Fanuc TP program (LS listing): JOB_VAR_COMMON.LS

/PROG  JOB_VAR_COMMON
/ATTR
OWNER		= MNEDITOR;
COMMENT		= "";
PROG_SIZE	= 43409;
CREATE		= DATE 19-03-19  TIME 16:19:56;
MODIFIED	= DATE 26-05-22  TIME 14:18:32;
FILE_NAME	= JOB_VAR_;
VERSION		= 0;
LINE_COUNT	= 1720;
MEMORY_SIZE	= 43957;
PROTECT		= READ_WRITE;
TCD:  STACK_SIZE	= 0,
      TASK_PRIORITY	= 50,
      TIME_SLICE	= 0,
      BUSY_LAMP_OFF	= 0,
      ABORT_REQUEST	= 0,
      PAUSE_REQUEST	= 0;
DEFAULT_GROUP	= 1,*,*,*,*;
CONTROL_CODE	= 00000000 00000000;
/APPL

AUTO_SINGULARITY_HEADER;
  ENABLE_SINGULARITY_AVOIDANCE   : TRUE;
/MN
   1:  !This is the common point ;
   2:  !template, all points are ;
   3:  !same if concentric ;
   4:  !---------------------------- ;
   5:  !Assign variable point profile ;
   6:  R[103]=AR[1]    ;
   7:  !--------------------------- ;
   8:  !SR[1] = "JOB_VAR_ID_GRIP" ;
   9:  !R[103]=100 -> "JOB_VAR_ID_GRIP" ;
  10:  !---------------------------- ;
  11:  !2By3 INF ID-GRIP, Max 18 piece ;
  12:  !Straight Face-plate Up/Down Pick ;
  13:  !---------------------------- ;
  14:  SELECT R[103]=100,JMP LBL[100] ;
  15:  !---------------------------- ;
  16:  !2By3 INF ID-GRIP, 45Deg Shift ;
  17:  !J4 Shift to Diagonal Pick ;
  18:         =110,JMP LBL[110] ;
  19:  !---------------------------- ;
  20:  !3By4 INF Sheet, Max 36 piece ;
  21:  !Straight Face-plate Up/Down Pick ;
  22:         =150,JMP LBL[150] ;
  23:  !---------------------------- ;
  24:  !3By4 INF Sheet, metal plate Max ;
  25:  !Straight Face-plate Up/Down Pick ;
  26:         =160,JMP LBL[160] ;
  27:  !---------------------------- ;
  28:  !3By4 INF Sheet, Max 72 piece ;
  29:  !Straight Face-plate Up/Down Pick ;
  30:         =170,JMP LBL[170] ;
  31:  !---------------------------- ;
  32:  !SR[2] = "JOB_VAR_OD_GRIP" ;
  33:  !R[103]=200 -> "JOB_VAR_OD_GRIP" ;
  34:  !---------------------------- ;
  35:  !2By3 INF OD-GRIP, Max 18 piece ;
  36:  !Straight Face-plate Up/Down Pick ;
  37:         =200,JMP LBL[200] ;
  38:  !---------------------------- ;
  39:  !2By3 INF OD-GRIP, 45Deg Shift ;
  40:  !J4 Shift to Diagonal Pick ;
  41:         =210,JMP LBL[210] ;
  42:  !---------------------------- ;
  43:  !3By4 INF OD-GRIP, Max 36 piece ;
  44:  !Straight Face-plate Up/Down Pick ;
  45:         =250,JMP LBL[250] ;
  46:  !---------------------------- ;
  47:  !3By4 INF OD-GRIP, 45Deg Shift ;
  48:  !J4 Shift to Diagonal Pick ;
  49:         =260,JMP LBL[260] ;
  50:  !---------------------------- ;
  51:  !4By6 INF OD-GRIP, Max 144 piece ;
  52:  !6By9 OFT 3 Tray ;
  53:         =270,JMP LBL[270] ;
  54:  !---------------------------- ;
  55:  !4By6 INF OD-GRIP, Max 144 piece ;
  56:  !6By8 OFT 3 Tray ;
  57:         =280,JMP LBL[280] ;
  58:  !---------------------------- ;
  59:  !Bar Feed OFT only, Max 144 piece ;
  60:  !4By9 OFT 4 Tray ;
  61:         =300,JMP LBL[300] ;
  62:  !---------------------------- ;
  63:  !Bar Feed OFT only, Max 144 piece ;
  64:  !6By8 OFT 3 Tray ;
  65:         =320,JMP LBL[320] ;
  66:  !---------------------------- ;
  67:  !3By4 INF Box ;
  68:  !Straight Up/Down Pick ;
  69:         =340,JMP LBL[340] ;
  70:  !---------------------------- ;
  71:  LBL[100] ;
  72:  !---------------------------- ;
  73:  !R[103]=100 -> "JOB_VAR_ID_GRIP" ;
  74:  !2By3 INF ID-GRIP, Max 18 piece ;
  75:  !Straight Face-plate Up/Down Pick ;
  76:  !---------------------------- ;
  77:  !Built PR[40] as Infeed P[1] ;
  78:  R[200]=40    ;
  79:   ;
  80:  R[201]=120.088    ;
  81:  R[202]=782.289    ;
  82:  R[203]=500.058    ;
  83:  R[204]=(-150.905)    ;
  84:  R[205]=(-89.467)    ;
  85:  R[206]=(-28.099)    ;
  86:   ;
  87:  CALL CREATE_PR(R[200],R[201],R[202],R[203],R[204],R[205],R[206]) ;
  88:   ;
  89:  !---------------------------- ;
  90:  !R[103]=100 -> "JOB_VAR_ID_GRIP" ;
  91:  !2By3 INF ID-GRIP, Max 18 piece ;
  92:  !Straight Face-plate Up/Down Pick ;
  93:  !---------------------------- ;
  94:  !Built PR[41] as Infeed P[2] ;
  95:  R[210]=41    ;
  96:   ;
  97:  R[211]=120.251    ;
  98:  R[212]=334.967    ;
  99:  R[213]=500.04    ;
 100:  R[214]=(-147.763)    ;
 101:  R[215]=(-89.089)    ;
 102:  R[216]=(-31.313)    ;
 103:   ;
 104:  CALL CREATE_PR(R[210],R[211],R[212],R[213],R[214],R[215],R[216]) ;
 105:   ;
 106:  !---------------------------- ;
 107:  !R[103]=100 -> "JOB_VAR_ID_GRIP" ;
 108:  !2By3 INF ID-GRIP, Max 18 piece ;
 109:  !Straight Face-plate Up/Down Pick ;
 110:  !---------------------------- ;
 111:  !Built PR[42] as Infeed P[3] ;
 112:  R[220]=42    ;
 113:   ;
 114:  R[221]=118.765    ;
 115:  R[222]=(-120.642)    ;
 116:  R[223]=500.756    ;
 117:  R[224]=(-153.606)    ;
 118:  R[225]=(-89.098)    ;
 119:  R[226]=(-25.398)    ;
 120:   ;
 121:  CALL CREATE_PR(R[220],R[221],R[222],R[223],R[224],R[225],R[226]) ;
 122:   ;
 123:  !---------------------------- ;
 124:  !R[103]=100 -> "JOB_VAR_ID_GRIP" ;
 125:  !2By3 INF ID-GRIP, Max 18 piece ;
 126:  !Straight Face-plate Up/Down Pick ;
 127:  !---------------------------- ;
 128:  !Built PR[50] as Outfeed P[1] ;
 129:  R[230]=50    ;
 130:   ;
 131:  R[231]=110.122    ;
 132:  R[232]=(-117.756)    ;
 133:  R[233]=500    ;
 134:  R[234]=6.053    ;
 135:  R[235]=(-88.646)    ;
 136:  R[236]=173.167    ;
 137:   ;
 138:  CALL CREATE_PR(R[230],R[231],R[232],R[233],R[234],R[235],R[236]) ;
 139:   ;
 140:  !---------------------------- ;
 141:  !R[103]=100 -> "JOB_VAR_ID_GRIP" ;
 142:  !2By3 INF ID-GRIP, Max 18 piece ;
 143:  !Straight Face-plate Up/Down Pick ;
 144:  !---------------------------- ;
 145:  !Built PR[51] as Outfeed P[2] ;
 146:  R[240]=51    ;
 147:   ;
 148:  R[241]=113.046    ;
 149:  R[242]=333.772    ;
 150:  R[243]=500    ;
 151:  R[244]=5.59    ;
 152:  R[245]=(-88.801)    ;
 153:  R[246]=173.593    ;
 154:   ;
 155:  CALL CREATE_PR(R[240],R[241],R[242],R[243],R[244],R[245],R[246]) ;
 156:   ;
 157:  !---------------------------- ;
 158:  !R[103]=100 -> "JOB_VAR_ID_GRIP" ;
 159:  !2By3 INF ID-GRIP, Max 18 piece ;
 160:  !Straight Face-plate Up/Down Pick ;
 161:  !---------------------------- ;
 162:  !Built PR[52] as Outfeed P[3] ;
 163:  R[250]=52    ;
 164:   ;
 165:  R[251]=115.343    ;
 166:  R[252]=785.028    ;
 167:  R[253]=500    ;
 168:  R[254]=(-7.342)    ;
 169:  R[255]=(-88.924)    ;
 170:  R[256]=(-173.386)    ;
 171:   ;
 172:  CALL CREATE_PR(R[250],R[251],R[252],R[253],R[254],R[255],R[256]) ;
 173:   ;
 174:  !Jump to end of the program ;
 175:  JMP LBL[9999] ;
 176:  !Template Ends ;
 177:   ;
 178:  !---------------------------- ;
 179:  LBL[110] ;
 180:  !---------------------------- ;
 181:  !R[103]=110 -> "JOB_VAR_ID_GRIP" ;
 182:  !2By3 INF ID-GRIP, 45Deg Shift ;
 183:  !J4 Shift to Diagonal Pick ;
 184:  !---------------------------- ;
 185:  !2By3 INF ID-GRIP, Max 18 piece ;
 186:  !---------------------------- ;
 187:  !Built PR[40] as Infeed P[1] ;
 188:  R[200]=40    ;
 189:   ;
 190:  R[201]=112.509    ;
 191:  R[202]=779.307    ;
 192:  R[203]=300    ;
 193:  R[204]=148.582    ;
 194:  R[205]=(-89.868)    ;
 195:  R[206]=(-7.553)    ;
 196:   ;
 197:  CALL CREATE_PR(R[200],R[201],R[202],R[203],R[204],R[205],R[206]) ;
 198:   ;
 199:  !---------------------------- ;
 200:  !R[103]=110 -> "JOB_VAR_ID_GRIP" ;
 201:  !2By3 INF ID-GRIP, 45Deg Shift ;
 202:  !J4 Shift to Diagonal Pick ;
 203:  !---------------------------- ;
 204:  !Built PR[41] as Infeed P[2] ;
 205:  R[210]=41    ;
 206:   ;
 207:  R[211]=112.917    ;
 208:  R[212]=329.437    ;
 209:  R[213]=300    ;
 210:  R[214]=157.871    ;
 211:  R[215]=(-89.833)    ;
 212:  R[216]=(-16.841)    ;
 213:   ;
 214:  CALL CREATE_PR(R[210],R[211],R[212],R[213],R[214],R[215],R[216]) ;
 215:   ;
 216:  !---------------------------- ;
 217:  !R[103]=110 -> "JOB_VAR_ID_GRIP" ;
 218:  !2By3 INF ID-GRIP, 45Deg Shift ;
 219:  !J4 Shift to Diagonal Pick ;
 220:  !---------------------------- ;
 221:  !Built PR[42] as Infeed P[3] ;
 222:  R[220]=42    ;
 223:   ;
 224:  R[221]=112.976    ;
 225:  R[222]=(-121.647)    ;
 226:  R[223]=300    ;
 227:  R[224]=162.478    ;
 228:  R[225]=(-89.805)    ;
 229:  R[226]=(-21.447)    ;
 230:   ;
 231:  CALL CREATE_PR(R[220],R[221],R[222],R[223],R[224],R[225],R[226]) ;
 232:   ;
 233:  !---------------------------- ;
 234:  !R[103]=110 -> "JOB_VAR_ID_GRIP" ;
 235:  !2By3 INF ID-GRIP, 45Deg Shift ;
 236:  !J4 Shift to Diagonal Drop ;
 237:  !---------------------------- ;
 238:  !Built PR[50] as OTF P[1] ;
 239:  R[230]=50    ;
 240:   ;
 241:  R[231]=110.895    ;
 242:  R[232]=(-123.626)    ;
 243:  R[233]=300    ;
 244:  R[234]=155.317    ;
 245:  R[235]=(-89.484)    ;
 246:  R[236]=(-24.715)    ;
 247:   ;
 248:  CALL CREATE_PR(R[230],R[231],R[232],R[233],R[234],R[235],R[236]) ;
 249:   ;
 250:  !---------------------------- ;
 251:  !R[103]=110 -> "JOB_VAR_ID_GRIP" ;
 252:  !2By3 INF ID-GRIP, 45Deg Shift ;
 253:  !J4 Shift to Diagonal Drop ;
 254:  !---------------------------- ;
 255:  !Built PR[51] as OTF P[2] ;
 256:  R[240]=51    ;
 257:   ;
 258:  R[241]=112.415    ;
 259:  R[242]=326.508    ;
 260:  R[243]=300    ;
 261:  R[244]=156.037    ;
 262:  R[245]=(-89.475)    ;
 263:  R[246]=(-25.441)    ;
 264:   ;
 265:  CALL CREATE_PR(R[240],R[241],R[242],R[243],R[244],R[245],R[246]) ;
 266:   ;
 267:  !---------------------------- ;
 268:  !R[103]=110 -> "JOB_VAR_ID_GRIP" ;
 269:  !2By3 INF ID-GRIP, 45Deg Shift ;
 270:  !J4 Shift to Diagonal Drop ;
 271:  !---------------------------- ;
 272:  !Built PR[52] as OTF P[3] ;
 273:  R[250]=52    ;
 274:   ;
 275:  R[251]=113.171    ;
 276:  R[252]=777.28    ;
 277:  R[253]=300    ;
 278:  R[254]=155.207    ;
 279:  R[255]=(-89.455)    ;
 280:  R[256]=(-24.623)    ;
 281:   ;
 282:  CALL CREATE_PR(R[250],R[251],R[252],R[253],R[254],R[255],R[256]) ;
 283:   ;
 284:  !Jump to end of the program ;
 285:  JMP LBL[9999] ;
 286:  !Template Ends ;
 287:   ;
 288:  !---------------------------- ;
 289:  LBL[150] ;
 290:  !---------------------------- ;
 291:  !R[103]=150 -> "JOB_VAR_ID_GRIP" ;
 292:  !3By4 INF Sheet, Max 36 piece ;
 293:  !Straight Face-plate Up/Down Pick ;
 294:  !---------------------------- ;
 295:  !Built PR[40] as Infeed P[1] ;
 296:  R[200]=40    ;
 297:   ;
 298:  R[201]=69.764    ;
 299:  R[202]=828.432    ;
 300:  R[203]=300    ;
 301:  R[204]=(-158.565)    ;
 302:  R[205]=(-89.413)    ;
 303:  R[206]=(-20.581)    ;
 304:   ;
 305:  CALL CREATE_PR(R[200],R[201],R[202],R[203],R[204],R[205],R[206]) ;
 306:   ;
 307:  !---------------------------- ;
 308:  !R[103]=150 -> "JOB_VAR_ID_GRIP" ;
 309:  !Straight Up/Down Pick ;
 310:  !3By4 INF Sheet, Max 36 piece ;
 311:  !---------------------------- ;
 312:  !Built PR[41] as Infeed P[2] ;
 313:  R[210]=41    ;
 314:   ;
 315:  R[211]=72.484    ;
 316:  R[212]=376.905    ;
 317:  R[213]=300    ;
 318:  R[214]=(-149.34)    ;
 319:  R[215]=(-89.283)    ;
 320:  R[216]=(-29.779)    ;
 321:   ;
 322:  CALL CREATE_PR(R[210],R[211],R[212],R[213],R[214],R[215],R[216]) ;
 323:   ;
 324:  !---------------------------- ;
 325:  !R[103]=150 -> "JOB_VAR_ID_GRIP" ;
 326:  !3By4 INF Sheet, Max 36 piece ;
 327:  !Straight Face-plate Up/Down Pick ;
 328:  !---------------------------- ;
 329:  !Built PR[42] as Infeed P[3] ;
 330:  R[220]=42    ;
 331:   ;
 332:  R[221]=73.047    ;
 333:  R[222]=(-73.901)    ;
 334:  R[223]=300    ;
 335:  R[224]=(-162.774)    ;
 336:  R[225]=(-88.893)    ;
 337:  R[226]=(-16.221)    ;
 338:   ;
 339:  CALL CREATE_PR(R[220],R[221],R[222],R[223],R[224],R[225],R[226]) ;
 340:   ;
 341:  !---------------------------- ;
 342:  !R[103]=150 -> "JOB_VAR_ID_GRIP" ;
 343:  !3By4 INF Sheet, Max 36 piece ;
 344:  !Straight Face-plate Up/Down Pick ;
 345:  !---------------------------- ;
 346:  !Built PR[50] as OTF P[1] ;
 347:  R[230]=50    ;
 348:   ;
 349:  R[231]=66.596    ;
 350:  R[232]=(-72.932)    ;
 351:  R[233]=300    ;
 352:  R[234]=5.353    ;
 353:  R[235]=(-88.806)    ;
 354:  R[236]=173.83    ;
 355:   ;
 356:  CALL CREATE_PR(R[230],R[231],R[232],R[233],R[234],R[235],R[236]) ;
 357:   ;
 358:  !---------------------------- ;
 359:  !R[103]=150 -> "JOB_VAR_ID_GRIP" ;
 360:  !3By4 INF Sheet, Max 36 piece ;
 361:  !Straight Face-plate Up/Down Pick ;
 362:  !---------------------------- ;
 363:  !Built PR[51] as OTF P[2] ;
 364:  R[240]=51    ;
 365:   ;
 366:  R[241]=70.095    ;
 367:  R[242]=378.905    ;
 368:  R[243]=300    ;
 369:  R[244]=(-4.178)    ;
 370:  R[245]=(-88.742)    ;
 371:  R[246]=(-176.605)    ;
 372:   ;
 373:  CALL CREATE_PR(R[240],R[241],R[242],R[243],R[244],R[245],R[246]) ;
 374:   ;
 375:  !---------------------------- ;
 376:  !R[103]=150 -> "JOB_VAR_ID_GRIP" ;
 377:  !3By4 INF Sheet, Max 36 piece ;
 378:  !Straight Face-plate Up/Down Pick ;
 379:  !---------------------------- ;
 380:  !Built PR[52] as OTF P[3] ;
 381:  R[250]=52    ;
 382:   ;
 383:  R[251]=70.211    ;
 384:  R[252]=829.862    ;
 385:  R[253]=300    ;
 386:  R[254]=(-7.014)    ;
 387:  R[255]=(-88.859)    ;
 388:  R[256]=(-173.67)    ;
 389:   ;
 390:  CALL CREATE_PR(R[250],R[251],R[252],R[253],R[254],R[255],R[256]) ;
 391:   ;
 392:  !Jump to end of the program ;
 393:  JMP LBL[9999] ;
 394:  !Template Ends ;
 395:   ;
 396:  !---------------------------- ;
 397:  LBL[160] ;
 398:  !---------------------------- ;
 399:  !R[103]=160 -> "JOB_VAR_ID_GRIP" ;
 400:  !3By4 INF Sheet, metal plate Max ;
 401:  !Straight Face-plate Up/Down Pick ;
 402:  !---------------------------- ;
 403:  !Built PR[40] as Infeed P[1] ;
 404:  R[200]=40    ;
 405:   ;
 406:  R[201]=78.195    ;
 407:  R[202]=824.843    ;
 408:  R[203]=300    ;
 409:  R[204]=(-.36)    ;
 410:  R[205]=(-88.464)    ;
 411:  R[206]=(-178.776)    ;
 412:   ;
 413:  CALL CREATE_PR(R[200],R[201],R[202],R[203],R[204],R[205],R[206]) ;
 414:   ;
 415:  !---------------------------- ;
 416:  !R[103]=160 -> "JOB_VAR_ID_GRIP" ;
 417:  !3By4 INF Sheet, metal plate Max ;
 418:  !Straight Face-plate Up/Down Pick ;
 419:  !---------------------------- ;
 420:  !Built PR[41] as Infeed P[2] ;
 421:  R[210]=41    ;
 422:   ;
 423:  R[211]=75.096    ;
 424:  R[212]=376.135    ;
 425:  R[213]=300    ;
 426:  R[214]=24.515    ;
 427:  R[215]=(-88.736)    ;
 428:  R[216]=156.675    ;
 429:   ;
 430:  CALL CREATE_PR(R[210],R[211],R[212],R[213],R[214],R[215],R[216]) ;
 431:   ;
 432:  !---------------------------- ;
 433:  !R[103]=160 -> "JOB_VAR_ID_GRIP" ;
 434:  !3By4 INF Sheet, metal plate Max ;
 435:  !Straight Face-plate Up/Down Pick ;
 436:  !---------------------------- ;
 437:  !Built PR[42] as Infeed P[3] ;
 438:  R[220]=42    ;
 439:   ;
 440:  R[221]=72.884    ;
 441:  R[222]=(-76.019)    ;
 442:  R[223]=300    ;
 443:  R[224]=(-1.211)    ;
 444:  R[225]=(-88.387)    ;
 445:  R[226]=(-177.625)    ;
 446:   ;
 447:  CALL CREATE_PR(R[220],R[221],R[222],R[223],R[224],R[225],R[226]) ;
 448:   ;
 449:  !---------------------------- ;
 450:  !R[103]=160 -> "JOB_VAR_ID_GRIP" ;
 451:  !3By4 INF Sheet, metal plate Max ;
 452:  !Straight Face-plate Up/Down Pick ;
 453:  !---------------------------- ;
 454:  !Built PR[50] as OTF P[1] ;
 455:  R[230]=50    ;
 456:   ;
 457:  R[231]=66.596    ;
 458:  R[232]=(-72.932)    ;
 459:  R[233]=700    ;
 460:  R[234]=5.353    ;
 461:  R[235]=(-88.806)    ;
 462:  R[236]=173.83    ;
 463:   ;
 464:  CALL CREATE_PR(R[230],R[231],R[232],R[233],R[234],R[235],R[236]) ;
 465:   ;
 466:  !---------------------------- ;
 467:  !R[103]=160 -> "JOB_VAR_ID_GRIP" ;
 468:  !3By4 INF Sheet, metal plate Max ;
 469:  !Straight Face-plate Up/Down Pick ;
 470:  !---------------------------- ;
 471:  !Built PR[51] as OTF P[2] ;
 472:  R[240]=51    ;
 473:   ;
 474:  R[241]=70.095    ;
 475:  R[242]=378.905    ;
 476:  R[243]=700    ;
 477:  R[244]=(-4.178)    ;
 478:  R[245]=(-88.742)    ;
 479:  R[246]=(-176.605)    ;
 480:   ;
 481:  CALL CREATE_PR(R[240],R[241],R[242],R[243],R[244],R[245],R[246]) ;
 482:   ;
 483:  !---------------------------- ;
 484:  !R[103]=160 -> "JOB_VAR_ID_GRIP" ;
 485:  !3By4 INF Sheet, metal plate Max ;
 486:  !Straight Face-plate Up/Down Pick ;
 487:  !---------------------------- ;
 488:  !Built PR[52] as OTF P[3] ;
 489:  R[250]=52    ;
 490:   ;
 491:  R[251]=70.211    ;
 492:  R[252]=829.862    ;
 493:  R[253]=700    ;
 494:  R[254]=(-7.014)    ;
 495:  R[255]=(-88.859)    ;
 496:  R[256]=(-173.67)    ;
 497:   ;
 498:  CALL CREATE_PR(R[250],R[251],R[252],R[253],R[254],R[255],R[256]) ;
 499:   ;
 500:  !Jump to end of the program ;
 501:  JMP LBL[9999] ;
 502:  !Template Ends ;
 503:   ;
 504:  !---------------------------- ;
 505:  LBL[170] ;
 506:  !---------------------------- ;
 507:  !R[103]=170 -> "JOB_VAR_ID_GRIP" ;
 508:  !3By4 INF Sheet, Max 72 piece ;
 509:  !Straight Face-plate Up/Down Pick ;
 510:  !---------------------------- ;
 511:  !Built PR[40] as Infeed P[1] ;
 512:  R[200]=40    ;
 513:   ;
 514:  R[201]=70.947    ;
 515:  R[202]=827.937    ;
 516:  R[203]=300    ;
 517:  R[204]=19.09    ;
 518:  R[205]=(-88.606)    ;
 519:  R[206]=161.741    ;
 520:   ;
 521:  CALL CREATE_PR(R[200],R[201],R[202],R[203],R[204],R[205],R[206]) ;
 522:   ;
 523:  !---------------------------- ;
 524:  !R[103]=170 -> "JOB_VAR_ID_GRIP" ;
 525:  !3By4 INF Sheet, Max 72 piece ;
 526:  !Straight Face-plate Up/Down Pick ;
 527:  !---------------------------- ;
 528:  !Built PR[41] as Infeed P[2] ;
 529:  R[210]=41    ;
 530:   ;
 531:  R[211]=69.577    ;
 532:  R[212]=378.246    ;
 533:  R[213]=300    ;
 534:  R[214]=19.393    ;
 535:  R[215]=(-88.529)    ;
 536:  R[216]=161.453    ;
 537:   ;
 538:  CALL CREATE_PR(R[210],R[211],R[212],R[213],R[214],R[215],R[216]) ;
 539:   ;
 540:  !---------------------------- ;
 541:  !R[103]=170 -> "JOB_VAR_ID_GRIP" ;
 542:  !3By4 INF Sheet, Max 72 piece ;
 543:  !Straight Face-plate Up/Down Pick ;
 544:  !---------------------------- ;
 545:  !Built PR[42] as Infeed P[3] ;
 546:  R[220]=42    ;
 547:   ;
 548:  R[221]=67.051    ;
 549:  R[222]=(-70.861)    ;
 550:  R[223]=300    ;
 551:  R[224]=17.005    ;
 552:  R[225]=(-88.405)    ;
 553:  R[226]=163.867    ;
 554:   ;
 555:  CALL CREATE_PR(R[220],R[221],R[222],R[223],R[224],R[225],R[226]) ;
 556:   ;
 557:  !---------------------------- ;
 558:  !R[103]=170 -> "JOB_VAR_ID_GRIP" ;
 559:  !3By4 INF Sheet, Max 72 piece ;
 560:  !Straight Face-plate Up/Down Pick ;
 561:  !---------------------------- ;
 562:  !Built PR[46] as Infeed P[4] ;
 563:  R[230]=46    ;
 564:   ;
 565:  R[231]=66.596    ;
 566:  R[232]=(-72.932)    ;
 567:  R[233]=300    ;
 568:  R[234]=5.353    ;
 569:  R[235]=(-88.806)    ;
 570:  R[236]=173.83    ;
 571:   ;
 572:  CALL CREATE_PR(R[230],R[231],R[232],R[233],R[234],R[235],R[236]) ;
 573:   ;
 574:  !---------------------------- ;
 575:  !R[103]=170 -> "JOB_VAR_ID_GRIP" ;
 576:  !3By4 INF Sheet, Max 72 piece ;
 577:  !Straight Face-plate Up/Down Pick ;
 578:  !---------------------------- ;
 579:  !Built PR[47] as Infeed P[5] ;
 580:  R[240]=47    ;
 581:   ;
 582:  R[241]=70.095    ;
 583:  R[242]=378.905    ;
 584:  R[243]=300    ;
 585:  R[244]=(-4.178)    ;
 586:  R[245]=(-88.742)    ;
 587:  R[246]=(-176.605)    ;
 588:   ;
 589:  CALL CREATE_PR(R[240],R[241],R[242],R[243],R[244],R[245],R[246]) ;
 590:   ;
 591:  !---------------------------- ;
 592:  !R[103]=170 -> "JOB_VAR_ID_GRIP" ;
 593:  !3By4 INF Sheet, Max 72 piece ;
 594:  !Straight Face-plate Up/Down Pick ;
 595:  !---------------------------- ;
 596:  !Built PR[48] as Infeed P[6] ;
 597:  R[250]=48    ;
 598:   ;
 599:  R[251]=70.211    ;
 600:  R[252]=829.862    ;
 601:  R[253]=300    ;
 602:  R[254]=(-7.014)    ;
 603:  R[255]=(-88.859)    ;
 604:  R[256]=(-173.67)    ;
 605:   ;
 606:  CALL CREATE_PR(R[250],R[251],R[252],R[253],R[254],R[255],R[256]) ;
 607:   ;
 608:  !---------------------------- ;
 609:  !R[103]=170 -> "JOB_VAR_ID_GRIP" ;
 610:  !3By4 INF Sheet, Max 72 piece ;
 611:  !Straight Face-plate Up/Down Pick ;
 612:  !---------------------------- ;
 613:  !Built PR[50] as OTF P[1] ;
 614:  R[260]=50    ;
 615:   ;
 616:  R[261]=32.757    ;
 617:  R[262]=214.942    ;
 618:  R[263]=300    ;
 619:  R[264]=(-157.549)    ;
 620:  R[265]=(-88.385)    ;
 621:  R[266]=(-19.293)    ;
 622:   ;
 623:  CALL CREATE_PR(R[260],R[261],R[262],R[263],R[264],R[265],R[266]) ;
 624:   ;
 625:  !---------------------------- ;
 626:  !R[103]=170 -> "JOB_VAR_ID_GRIP" ;
 627:  !3By4 INF Sheet, Max 72 piece ;
 628:  !Straight Face-plate Up/Down Pick ;
 629:  !---------------------------- ;
 630:  !Built PR[51] as OTF P[2] ;
 631:  R[270]=51    ;
 632:   ;
 633:  R[271]=33.41    ;
 634:  R[272]=503.872    ;
 635:  R[273]=300    ;
 636:  R[274]=(-157.614)    ;
 637:  R[275]=(-88.378)    ;
 638:  R[276]=(-19.237)    ;
 639:   ;
 640:  CALL CREATE_PR(R[270],R[271],R[272],R[273],R[274],R[275],R[276]) ;
 641:   ;
 642:  !---------------------------- ;
 643:  !R[103]=170 -> "JOB_VAR_ID_GRIP" ;
 644:  !3By4 INF Sheet, Max 72 piece ;
 645:  !Straight Face-plate Up/Down Pick ;
 646:  !---------------------------- ;
 647:  !Built PR[52] as OTF P[3] ;
 648:  R[280]=52    ;
 649:   ;
 650:  R[281]=34.713    ;
 651:  R[282]=788.151    ;
 652:  R[283]=300    ;
 653:  R[284]=(-157.828)    ;
 654:  R[285]=(-88.37)    ;
 655:  R[286]=(-19.031)    ;
 656:   ;
 657:  CALL CREATE_PR(R[280],R[281],R[282],R[283],R[284],R[285],R[286]) ;
 658:   ;
 659:  !---------------------------- ;
 660:  !R[103]=170 -> "JOB_VAR_ID_GRIP" ;
 661:  !3By4 INF Sheet, Max 72 piece ;
 662:  !Straight Face-plate Up/Down Pick ;
 663:  !---------------------------- ;
 664:  !Built PR[60] as OTF P[4] ;
 665:  R[290]=60    ;
 666:   ;
 667:  R[291]=30.529    ;
 668:  R[292]=1075.31    ;
 669:  R[293]=300    ;
 670:  R[294]=(-157.993)    ;
 671:  R[295]=(-88.367)    ;
 672:  R[296]=(-18.874)    ;
 673:   ;
 674:  CALL CREATE_PR(R[290],R[291],R[292],R[293],R[294],R[295],R[296]) ;
 675:   ;
 676:  !Jump to end of the program ;
 677:  JMP LBL[9999] ;
 678:  !Template Ends ;
 679:   ;
 680:  !---------------------------- ;
 681:  LBL[200] ;
 682:  !---------------------------- ;
 683:  !R[103]=200 -> "JOB_VAR_OD_GRIP" ;
 684:  !2By3 INF OD-GRIP, Max 18 piece ;
 685:  !Straight Face-plate Up/Down Pick ;
 686:  !---------------------------- ;
 687:  !Built PR[40] as Infeed P[1] ;
 688:  R[200]=40    ;
 689:   ;
 690:  R[201]=112.982    ;
 691:  R[202]=784.424    ;
 692:  R[203]=500    ;
 693:  R[204]=(-126.216)    ;
 694:  R[205]=(-89.241)    ;
 695:  R[206]=(-52.902)    ;
 696:   ;
 697:  CALL CREATE_PR(R[200],R[201],R[202],R[203],R[204],R[205],R[206]) ;
 698:   ;
 699:  !---------------------------- ;
 700:  !R[103]=200 -> "JOB_VAR_OD_GRIP" ;
 701:  !2By3 INF OD-GRIP, Max 18 piece ;
 702:  !Straight Face-plate Up/Down Pick ;
 703:  !---------------------------- ;
 704:  !Built PR[41] as Infeed P[2] ;
 705:  R[210]=41    ;
 706:   ;
 707:  R[211]=115.261    ;
 708:  R[212]=333.579    ;
 709:  R[213]=500    ;
 710:  R[214]=(-129.455)    ;
 711:  R[215]=(-89.194)    ;
 712:  R[216]=(-49.607)    ;
 713:   ;
 714:  CALL CREATE_PR(R[210],R[211],R[212],R[213],R[214],R[215],R[216]) ;
 715:   ;
 716:  !---------------------------- ;
 717:  !R[103]=200 -> "JOB_VAR_OD_GRIP" ;
 718:  !2By3 INF OD-GRIP, Max 18 piece ;
 719:  !Straight Face-plate Up/Down Pick ;
 720:  !---------------------------- ;
 721:  !Built PR[42] as Infeed P[3] ;
 722:  R[220]=42    ;
 723:   ;
 724:  R[221]=117.201    ;
 725:  R[222]=(-118.434)    ;
 726:  R[223]=500    ;
 727:  R[224]=(-140.645)    ;
 728:  R[225]=(-89.198)    ;
 729:  R[226]=(-38.372)    ;
 730:   ;
 731:  CALL CREATE_PR(R[220],R[221],R[222],R[223],R[224],R[225],R[226]) ;
 732:   ;
 733:  !---------------------------- ;
 734:  !R[103]=200 -> "JOB_VAR_OD_GRIP" ;
 735:  !2By3 INF OD-GRIP, Max 18 piece ;
 736:  !Straight Face-plate Up/Down Pick ;
 737:  !---------------------------- ;
 738:  !Built PR[50] as Outfeed P[1] ;
 739:  R[230]=50    ;
 740:   ;
 741:  R[231]=110.061    ;
 742:  R[232]=(-117.791)    ;
 743:  R[233]=500    ;
 744:  R[234]=(-132.147)    ;
 745:  R[235]=(-89.011)    ;
 746:  R[236]=(-48.619)    ;
 747:   ;
 748:  CALL CREATE_PR(R[230],R[231],R[232],R[233],R[234],R[235],R[236]) ;
 749:   ;
 750:  !---------------------------- ;
 751:  !R[103]=200 -> "JOB_VAR_OD_GRIP" ;
 752:  !2By3 INF OD-GRIP, Max 18 piece ;
 753:  !Straight Face-plate Up/Down Pick ;
 754:  !---------------------------- ;
 755:  !Built PR[51] as Outfeed P[2] ;
 756:  R[240]=51    ;
 757:   ;
 758:  R[241]=112.794    ;
 759:  R[242]=333.794    ;
 760:  R[243]=500    ;
 761:  R[244]=(-128.298)    ;
 762:  R[245]=(-89.118)    ;
 763:  R[246]=(-52.477)    ;
 764:   ;
 765:  CALL CREATE_PR(R[240],R[241],R[242],R[243],R[244],R[245],R[246]) ;
 766:   ;
 767:  !---------------------------- ;
 768:  !R[103]=200 -> "JOB_VAR_OD_GRIP" ;
 769:  !2By3 INF OD-GRIP, Max 18 piece ;
 770:  !Straight Face-plate Up/Down Pick ;
 771:  !---------------------------- ;
 772:  !Built PR[52] as Outfeed P[3] ;
 773:  R[250]=52    ;
 774:   ;
 775:  R[251]=114.882    ;
 776:  R[252]=785.406    ;
 777:  R[253]=500    ;
 778:  R[254]=(-112.083)    ;
 779:  R[255]=(-89.23)    ;
 780:  R[256]=(-68.496)    ;
 781:   ;
 782:  CALL CREATE_PR(R[250],R[251],R[252],R[253],R[254],R[255],R[256]) ;
 783:   ;
 784:  !Jump to end of the program ;
 785:  JMP LBL[9999] ;
 786:  !Template Ends ;
 787:   ;
 788:  !---------------------------- ;
 789:  LBL[210] ;
 790:  !---------------------------- ;
 791:  !R[103]=210 -> "JOB_VAR_OD_GRIP" ;
 792:  !2By3 INF OD-GRIP, 45Deg Shift ;
 793:  !J4 Shift to Diagonal Pick ;
 794:  !---------------------------- ;
 795:  !Built PR[40] as Infeed P[1] ;
 796:  R[200]=40    ;
 797:   ;
 798:  R[201]=112.509    ;
 799:  R[202]=779.307    ;
 800:  R[203]=300    ;
 801:  R[204]=148.582    ;
 802:  R[205]=(-89.868)    ;
 803:  R[206]=(-7.553)    ;
 804:   ;
 805:  CALL CREATE_PR(R[200],R[201],R[202],R[203],R[204],R[205],R[206]) ;
 806:   ;
 807:  !---------------------------- ;
 808:  !R[103]=210 -> "JOB_VAR_OD_GRIP" ;
 809:  !2By3 INF OD-GRIP, 45Deg Shift ;
 810:  !J4 Shift to Diagonal Pick ;
 811:  !---------------------------- ;
 812:  !Built PR[41] as Infeed P[2] ;
 813:  R[210]=41    ;
 814:   ;
 815:  R[211]=112.917    ;
 816:  R[212]=329.437    ;
 817:  R[213]=300    ;
 818:  R[214]=157.871    ;
 819:  R[215]=(-89.833)    ;
 820:  R[216]=(-16.841)    ;
 821:   ;
 822:  CALL CREATE_PR(R[210],R[211],R[212],R[213],R[214],R[215],R[216]) ;
 823:   ;
 824:  !---------------------------- ;
 825:  !R[103]=210 -> "JOB_VAR_OD_GRIP" ;
 826:  !2By3 INF OD-GRIP, 45Deg Shift ;
 827:  !J4 Shift to Diagonal Pick ;
 828:  !---------------------------- ;
 829:  !Built PR[42] as Infeed P[3] ;
 830:  R[220]=42    ;
 831:   ;
 832:  R[221]=112.976    ;
 833:  R[222]=(-121.647)    ;
 834:  R[223]=300    ;
 835:  R[224]=162.478    ;
 836:  R[225]=(-89.805)    ;
 837:  R[226]=(-21.447)    ;
 838:   ;
 839:  CALL CREATE_PR(R[220],R[221],R[222],R[223],R[224],R[225],R[226]) ;
 840:   ;
 841:  !---------------------------- ;
 842:  !R[103]=210 -> "JOB_VAR_OD_GRIP" ;
 843:  !2By3 INF OD-GRIP, 45Deg Shift ;
 844:  !J4 Shift to Diagonal Pick ;
 845:  !---------------------------- ;
 846:  !Built PR[50] as OTF P[1] ;
 847:  R[230]=50    ;
 848:   ;
 849:  R[231]=110.895    ;
 850:  R[232]=(-123.626)    ;
 851:  R[233]=300    ;
 852:  R[234]=155.317    ;
 853:  R[235]=(-89.484)    ;
 854:  R[236]=(-24.715)    ;
 855:   ;
 856:  CALL CREATE_PR(R[230],R[231],R[232],R[233],R[234],R[235],R[236]) ;
 857:   ;
 858:  !---------------------------- ;
 859:  !R[103]=210 -> "JOB_VAR_OD_GRIP" ;
 860:  !2By3 INF OD-GRIP, 45Deg Shift ;
 861:  !J4 Shift to Diagonal Pick ;
 862:  !---------------------------- ;
 863:  !Built PR[51] as OTF P[2] ;
 864:  R[240]=51    ;
 865:   ;
 866:  R[241]=112.415    ;
 867:  R[242]=326.508    ;
 868:  R[243]=300    ;
 869:  R[244]=156.037    ;
 870:  R[245]=(-89.475)    ;
 871:  R[246]=(-25.441)    ;
 872:   ;
 873:  CALL CREATE_PR(R[240],R[241],R[242],R[243],R[244],R[245],R[246]) ;
 874:   ;
 875:  !---------------------------- ;
 876:  !R[103]=210 -> "JOB_VAR_OD_GRIP" ;
 877:  !2By3 INF OD-GRIP, 45Deg Shift ;
 878:  !J4 Shift to Diagonal Pick ;
 879:  !---------------------------- ;
 880:  !Built PR[52] as OTF P[3] ;
 881:  R[250]=52    ;
 882:   ;
 883:  R[251]=113.171    ;
 884:  R[252]=777.28    ;
 885:  R[253]=300    ;
 886:  R[254]=155.207    ;
 887:  R[255]=(-89.455)    ;
 888:  R[256]=(-24.623)    ;
 889:   ;
 890:  CALL CREATE_PR(R[250],R[251],R[252],R[253],R[254],R[255],R[256]) ;
 891:   ;
 892:  !Jump to end of the program ;
 893:  JMP LBL[9999] ;
 894:  !Template Ends ;
 895:   ;
 896:  !---------------------------- ;
 897:  LBL[250] ;
 898:  !---------------------------- ;
 899:  !R[103]=250 -> "JOB_VAR_OD_GRIP" ;
 900:  !3By4 INF OD-GRIP, Max 36 piece ;
 901:  !Straight Face-plate Up/Down Pick ;
 902:  !---------------------------- ;
 903:  !Built PR[40] as Infeed P[1] ;
 904:  R[200]=40    ;
 905:   ;
 906:  R[201]=70.947    ;
 907:  R[202]=827.937    ;
 908:  R[203]=300    ;
 909:  R[204]=19.09    ;
 910:  R[205]=(-88.606)    ;
 911:  R[206]=161.741    ;
 912:   ;
 913:  CALL CREATE_PR(R[200],R[201],R[202],R[203],R[204],R[205],R[206]) ;
 914:   ;
 915:  !---------------------------- ;
 916:  !R[103]=250 -> "JOB_VAR_OD_GRIP" ;
 917:  !3By4 INF OD-GRIP, Max 36 piece ;
 918:  !Straight Face-plate Up/Down Pick ;
 919:  !---------------------------- ;
 920:  !Built PR[41] as Infeed P[2] ;
 921:  R[210]=41    ;
 922:   ;
 923:  R[211]=69.577    ;
 924:  R[212]=378.246    ;
 925:  R[213]=300    ;
 926:  R[214]=19.393    ;
 927:  R[215]=(-88.529)    ;
 928:  R[216]=161.453    ;
 929:   ;
 930:  CALL CREATE_PR(R[210],R[211],R[212],R[213],R[214],R[215],R[216]) ;
 931:   ;
 932:  !---------------------------- ;
 933:  !R[103]=250 -> "JOB_VAR_OD_GRIP" ;
 934:  !3By4 INF OD-GRIP, Max 36 piece ;
 935:  !Straight Face-plate Up/Down Pick ;
 936:  !---------------------------- ;
 937:  !Built PR[42] as Infeed P[3] ;
 938:  R[220]=42    ;
 939:   ;
 940:  R[221]=67.051    ;
 941:  R[222]=(-70.861)    ;
 942:  R[223]=300    ;
 943:  R[224]=17.005    ;
 944:  R[225]=(-88.405)    ;
 945:  R[226]=163.867    ;
 946:   ;
 947:  CALL CREATE_PR(R[220],R[221],R[222],R[223],R[224],R[225],R[226]) ;
 948:   ;
 949:  !---------------------------- ;
 950:  !R[103]=250 -> "JOB_VAR_OD_GRIP" ;
 951:  !3By4 INF OD-GRIP, Max 36 piece ;
 952:  !Straight Face-plate Up/Down Pick ;
 953:  !---------------------------- ;
 954:  !Built PR[50] as OTF P[1] ;
 955:  R[230]=50    ;
 956:   ;
 957:  R[231]=66.596    ;
 958:  R[232]=(-72.932)    ;
 959:  R[233]=700    ;
 960:  R[234]=5.353    ;
 961:  R[235]=(-88.806)    ;
 962:  R[236]=173.83    ;
 963:   ;
 964:  CALL CREATE_PR(R[230],R[231],R[232],R[233],R[234],R[235],R[236]) ;
 965:   ;
 966:  !---------------------------- ;
 967:  !R[103]=250 -> "JOB_VAR_OD_GRIP" ;
 968:  !3By4 INF OD-GRIP, Max 36 piece ;
 969:  !Straight Face-plate Up/Down Pick ;
 970:  !---------------------------- ;
 971:  !Built PR[51] as OTF P[2] ;
 972:  R[240]=51    ;
 973:   ;
 974:  R[241]=70.095    ;
 975:  R[242]=378.905    ;
 976:  R[243]=700    ;
 977:  R[244]=(-4.178)    ;
 978:  R[245]=(-88.742)    ;
 979:  R[246]=(-176.605)    ;
 980:   ;
 981:  CALL CREATE_PR(R[240],R[241],R[242],R[243],R[244],R[245],R[246]) ;
 982:   ;
 983:  !---------------------------- ;
 984:  !R[103]=250 -> "JOB_VAR_OD_GRIP" ;
 985:  !3By4 INF OD-GRIP, Max 36 piece ;
 986:  !Straight Face-plate Up/Down Pick ;
 987:  !---------------------------- ;
 988:  !Built PR[52] as OTF P[3] ;
 989:  R[250]=52    ;
 990:   ;
 991:  R[251]=70.211    ;
 992:  R[252]=829.862    ;
 993:  R[253]=700    ;
 994:  R[254]=(-7.014)    ;
 995:  R[255]=(-88.859)    ;
 996:  R[256]=(-173.67)    ;
 997:   ;
 998:  CALL CREATE_PR(R[250],R[251],R[252],R[253],R[254],R[255],R[256]) ;
 999:   ;
1000:  !Jump to end of the program ;
1001:  JMP LBL[9999] ;
1002:  !Template Ends ;
1003:   ;
1004:  !---------------------------- ;
1005:  LBL[260] ;
1006:  !---------------------------- ;
1007:  !R[103]=260 -> "JOB_VAR_OD_GRIP" ;
1008:  !3By4 INF Sheet, Mandrel ;
1009:  !---------------------------- ;
1010:  !---------------------------- ;
1011:  !Built PR[40] as Infeed P[1] ;
1012:  R[200]=40    ;
1013:   ;
1014:  R[201]=80.718    ;
1015:  R[202]=822.937    ;
1016:  R[203]=700    ;
1017:  R[204]=(-168.381)    ;
1018:  R[205]=(-89.185)    ;
1019:  R[206]=(-12.041)    ;
1020:   ;
1021:  CALL CREATE_PR(R[200],R[201],R[202],R[203],R[204],R[205],R[206]) ;
1022:   ;
1023:  !---------------------------- ;
1024:  !R[103]=260 -> "JOB_VAR_OD_GRIP" ;
1025:  !3By4 INF OD-GRIP, Max 36 piece ;
1026:  !Straight Face-plate Up/Down Pick ;
1027:  !metal plate for mandrel ;
1028:  !---------------------------- ;
1029:  !Built PR[41] as Infeed P[2] ;
1030:  R[210]=41    ;
1031:   ;
1032:  R[211]=77.807    ;
1033:  R[212]=372.057    ;
1034:  R[213]=700    ;
1035:  R[214]=(-76.269)    ;
1036:  R[215]=(-89.693)    ;
1037:  R[216]=(-105.893)    ;
1038:   ;
1039:  CALL CREATE_PR(R[210],R[211],R[212],R[213],R[214],R[215],R[216]) ;
1040:   ;
1041:  !---------------------------- ;
1042:  !R[103]=260 -> "JOB_VAR_OD_GRIP" ;
1043:  !3By4 INF OD-GRIP, Max 36 piece ;
1044:  !Straight Face-plate Up/Down Pick ;
1045:  !metal plate for mandrel ;
1046:  !---------------------------- ;
1047:  !Built PR[50] as OTF P[1] ;
1048:  R[230]=50    ;
1049:   ;
1050:  R[231]=69.168    ;
1051:  R[232]=(-72.593)    ;
1052:  R[233]=800    ;
1053:  R[234]=(-156.246)    ;
1054:  R[235]=(-89.505)    ;
1055:  R[236]=(-23.868)    ;
1056:   ;
1057:  CALL CREATE_PR(R[230],R[231],R[232],R[233],R[234],R[235],R[236]) ;
1058:   ;
1059:  !---------------------------- ;
1060:  !R[103]=260 -> "JOB_VAR_OD_GRIP" ;
1061:  !3By4 INF OD-GRIP, Max 36 piece ;
1062:  !Straight Face-plate Up/Down Pick ;
1063:  !metal plate for mandrel ;
1064:  !---------------------------- ;
1065:  !Built PR[51] as OTF P[2] ;
1066:  R[240]=51    ;
1067:   ;
1068:  R[241]=68.548    ;
1069:  R[242]=377.148    ;
1070:  R[243]=800    ;
1071:  R[244]=(-155.546)    ;
1072:  R[245]=(-89.489)    ;
1073:  R[246]=(-24.568)    ;
1074:   ;
1075:  CALL CREATE_PR(R[240],R[241],R[242],R[243],R[244],R[245],R[246]) ;
1076:   ;
1077:  !Jump to end of the program ;
1078:  JMP LBL[9999] ;
1079:  !Template Ends ;
1080:   ;
1081:  LBL[270] ;
1082:  !---------------------------- ;
1083:  !R[103]=270 -> "JOB_VAR_OD_GRIP" ;
1084:  !4By6 INF OD-GRIP, Max 144 piece ;
1085:  !Straight Face-plate Up/Down Pick ;
1086:  !---------------------------- ;
1087:  !Built PR[40] as Infeed P[1] ;
1088:  R[200]=40    ;
1089:   ;
1090:  R[201]=52.986    ;
1091:  R[202]=837.611    ;
1092:  R[203]=300    ;
1093:  R[204]=(-135.64)    ;
1094:  R[205]=(-89.334)    ;
1095:  R[206]=(-44.75)    ;
1096:   ;
1097:  CALL CREATE_PR(R[200],R[201],R[202],R[203],R[204],R[205],R[206]) ;
1098:   ;
1099:  !---------------------------- ;
1100:  !R[103]=270 -> "JOB_VAR_OD_GRIP" ;
1101:  !4By6 INF OD-GRIP, Max 144 piece ;
1102:  !Straight Face-plate Up/Down Pick ;
1103:  !---------------------------- ;
1104:  !Built PR[41] as Infeed P[2] ;
1105:  R[210]=41    ;
1106:   ;
1107:  R[211]=53.152    ;
1108:  R[212]=385.263    ;
1109:  R[213]=300    ;
1110:  R[214]=(-136.806)    ;
1111:  R[215]=(-89.315)    ;
1112:  R[216]=(-43.565)    ;
1113:   ;
1114:  CALL CREATE_PR(R[210],R[211],R[212],R[213],R[214],R[215],R[216]) ;
1115:   ;
1116:  !---------------------------- ;
1117:  !R[103]=270 -> "JOB_VAR_OD_GRIP" ;
1118:  !4By6 INF OD-GRIP, Max 144 piece ;
1119:  !Straight Face-plate Up/Down Pick ;
1120:  !---------------------------- ;
1121:  !Built PR[42] as Infeed P[3] ;
1122:  R[220]=42    ;
1123:   ;
1124:  R[221]=44.932    ;
1125:  R[222]=357.144    ;
1126:  R[223]=300    ;
1127:  R[224]=(-127.616)    ;
1128:  R[225]=(-89.079)    ;
1129:  R[226]=(-52.124)    ;
1130:   ;
1131:  CALL CREATE_PR(R[220],R[221],R[222],R[223],R[224],R[225],R[226]) ;
1132:   ;
1133:  !---------------------------- ;
1134:  !R[103]=270 -> "JOB_VAR_OD_GRIP" ;
1135:  !4By6 INF OD-GRIP, Max 144 piece ;
1136:  !Straight Face-plate Up/Down Pick ;
1137:  !---------------------------- ;
1138:  !Built PR[47] as Infeed P[4] ;
1139:  R[230]=47    ;
1140:   ;
1141:  R[231]=53.084    ;
1142:  R[232]=836.564    ;
1143:  R[233]=300    ;
1144:  R[234]=(-127.701)    ;
1145:  R[235]=(-89.072)    ;
1146:  R[236]=(-53.116)    ;
1147:   ;
1148:  CALL CREATE_PR(R[230],R[231],R[232],R[233],R[234],R[235],R[236]) ;
1149:   ;
1150:  !---------------------------- ;
1151:  !R[103]=270 -> "JOB_VAR_OD_GRIP" ;
1152:  !4By6 INF OD-GRIP, Max 144 piece ;
1153:  !Straight Face-plate Up/Down Pick ;
1154:  !---------------------------- ;
1155:  !Built PR[48] as Infeed P[5] ;
1156:  R[240]=48    ;
1157:   ;
1158:  R[241]=53.598    ;
1159:  R[242]=386.354    ;
1160:  R[243]=300    ;
1161:  R[244]=(-119.135)    ;
1162:  R[245]=(-89.246)    ;
1163:  R[246]=(-62.104)    ;
1164:   ;
1165:  CALL CREATE_PR(R[240],R[241],R[242],R[243],R[244],R[245],R[246]) ;
1166:   ;
1167:  !---------------------------- ;
1168:  !R[103]=270 -> "JOB_VAR_OD_GRIP" ;
1169:  !4By6 INF OD-GRIP, Max 144 piece ;
1170:  !Straight Face-plate Up/Down Pick ;
1171:  !---------------------------- ;
1172:  !Built PR[49] as Infeed P[6] ;
1173:  R[250]=49    ;
1174:   ;
1175:  R[251]=52.953    ;
1176:  R[252]=(-59.846)    ;
1177:  R[253]=300    ;
1178:  R[254]=(-123.722)    ;
1179:  R[255]=(-89.153)    ;
1180:  R[256]=(-57.497)    ;
1181:   ;
1182:  CALL CREATE_PR(R[250],R[251],R[252],R[253],R[254],R[255],R[256]) ;
1183:   ;
1184:  !---------------------------- ;
1185:  !R[103]=270 -> "JOB_VAR_OD_GRIP" ;
1186:  !4By6 INF OD-GRIP, Max 144 piece ;
1187:  !Straight Face-plate Up/Down Pick ;
1188:  !---------------------------- ;
1189:  !Built PR[50] as OTF P[1] ;
1190:  R[260]=50    ;
1191:   ;
1192:  R[261]=32.757    ;
1193:  R[262]=214.942    ;
1194:  R[263]=300    ;
1195:  R[264]=(-157.549)    ;
1196:  R[265]=(-88.385)    ;
1197:  R[266]=(-19.293)    ;
1198:   ;
1199:  CALL CREATE_PR(R[260],R[261],R[262],R[263],R[264],R[265],R[266]) ;
1200:   ;
1201:  !---------------------------- ;
1202:  !R[103]=270 -> "JOB_VAR_OD_GRIP" ;
1203:  !4By6 INF OD-GRIP, Max 144 piece ;
1204:  !Straight Face-plate Up/Down Pick ;
1205:  !---------------------------- ;
1206:  !Built PR[51] as OTF P[2] ;
1207:  R[270]=51    ;
1208:   ;
1209:  R[271]=33.41    ;
1210:  R[272]=503.872    ;
1211:  R[273]=300    ;
1212:  R[274]=(-157.614)    ;
1213:  R[275]=(-88.378)    ;
1214:  R[276]=(-19.237)    ;
1215:   ;
1216:  CALL CREATE_PR(R[270],R[271],R[272],R[273],R[274],R[275],R[276]) ;
1217:   ;
1218:  !---------------------------- ;
1219:  !R[103]=270 -> "JOB_VAR_OD_GRIP" ;
1220:  !4By6 INF OD-GRIP, Max 144 piece ;
1221:  !Straight Face-plate Up/Down Pick ;
1222:  !---------------------------- ;
1223:  !Built PR[52] as OTF P[3] ;
1224:  R[280]=52    ;
1225:   ;
1226:  R[281]=34.713    ;
1227:  R[282]=788.151    ;
1228:  R[283]=300    ;
1229:  R[284]=(-157.828)    ;
1230:  R[285]=(-88.37)    ;
1231:  R[286]=(-19.031)    ;
1232:   ;
1233:  CALL CREATE_PR(R[280],R[281],R[282],R[283],R[284],R[285],R[286]) ;
1234:   ;
1235:  !---------------------------- ;
1236:  !R[103]=270 -> "JOB_VAR_OD_GRIP" ;
1237:  !4By6 INF OD-GRIP, Max 144 piece ;
1238:  !Straight Face-plate Up/Down Pick ;
1239:  !---------------------------- ;
1240:  !Built PR[60] as OTF P[4] ;
1241:  R[290]=60    ;
1242:   ;
1243:  R[291]=30.529    ;
1244:  R[292]=1075.31    ;
1245:  R[293]=300    ;
1246:  R[294]=(-157.993)    ;
1247:  R[295]=(-88.367)    ;
1248:  R[296]=(-18.874)    ;
1249:   ;
1250:  CALL CREATE_PR(R[290],R[291],R[292],R[293],R[294],R[295],R[296]) ;
1251:   ;
1252:  !Jump to end of the program ;
1253:  JMP LBL[9999] ;
1254:  !Template Ends ;
1255:   ;
1256:  !---------------------------- ;
1257:  LBL[280] ;
1258:  !---------------------------- ;
1259:  !Built PR[40] as Infeed P[1] ;
1260:  R[200]=40    ;
1261:   ;
1262:  R[201]=52.986    ;
1263:  R[202]=837.611    ;
1264:  R[203]=300    ;
1265:  R[204]=(-135.64)    ;
1266:  R[205]=(-89.334)    ;
1267:  R[206]=(-44.75)    ;
1268:   ;
1269:  CALL CREATE_PR(R[200],R[201],R[202],R[203],R[204],R[205],R[206]) ;
1270:   ;
1271:  !---------------------------- ;
1272:  !Built PR[41] as Infeed P[2] ;
1273:  R[210]=41    ;
1274:   ;
1275:  R[211]=53.152    ;
1276:  R[212]=385.263    ;
1277:  R[213]=300    ;
1278:  R[214]=(-136.806)    ;
1279:  R[215]=(-89.315)    ;
1280:  R[216]=(-43.565)    ;
1281:   ;
1282:  CALL CREATE_PR(R[210],R[211],R[212],R[213],R[214],R[215],R[216]) ;
1283:   ;
1284:  !---------------------------- ;
1285:  !Built PR[42] as Infeed P[3] ;
1286:  R[220]=42    ;
1287:   ;
1288:  R[221]=44.932    ;
1289:  R[222]=357.144    ;
1290:  R[223]=300    ;
1291:  R[224]=(-127.616)    ;
1292:  R[225]=(-89.079)    ;
1293:  R[226]=(-52.124)    ;
1294:   ;
1295:  CALL CREATE_PR(R[220],R[221],R[222],R[223],R[224],R[225],R[226]) ;
1296:   ;
1297:  !---------------------------- ;
1298:  !Built PR[47] as Infeed P[4] ;
1299:  R[230]=47    ;
1300:   ;
1301:  R[231]=53.084    ;
1302:  R[232]=836.564    ;
1303:  R[233]=300    ;
1304:  R[234]=(-127.701)    ;
1305:  R[235]=(-89.072)    ;
1306:  R[236]=(-53.116)    ;
1307:   ;
1308:  CALL CREATE_PR(R[230],R[231],R[232],R[233],R[234],R[235],R[236]) ;
1309:   ;
1310:  !---------------------------- ;
1311:  !Built PR[48] as Infeed P[5] ;
1312:  R[240]=48    ;
1313:   ;
1314:  R[241]=53.598    ;
1315:  R[242]=386.354    ;
1316:  R[243]=300    ;
1317:  R[244]=(-119.135)    ;
1318:  R[245]=(-89.246)    ;
1319:  R[246]=(-62.104)    ;
1320:   ;
1321:  CALL CREATE_PR(R[240],R[241],R[242],R[243],R[244],R[245],R[246]) ;
1322:   ;
1323:  !---------------------------- ;
1324:  !Built PR[49] as Infeed P[6] ;
1325:  R[250]=49    ;
1326:   ;
1327:  R[251]=52.953    ;
1328:  R[252]=(-59.846)    ;
1329:  R[253]=300    ;
1330:  R[254]=(-123.722)    ;
1331:  R[255]=(-89.153)    ;
1332:  R[256]=(-57.497)    ;
1333:   ;
1334:  CALL CREATE_PR(R[250],R[251],R[252],R[253],R[254],R[255],R[256]) ;
1335:   ;
1336:  !---------------------------- ;
1337:  !Built PR[50] as OTF P[1] ;
1338:  R[260]=50    ;
1339:   ;
1340:  R[261]=57.682    ;
1341:  R[262]=(-63.727)    ;
1342:  R[263]=300    ;
1343:  R[264]=(-171.541)    ;
1344:  R[265]=(-88.207)    ;
1345:  R[266]=(-7.451)    ;
1346:   ;
1347:  CALL CREATE_PR(R[260],R[261],R[262],R[263],R[264],R[265],R[266]) ;
1348:   ;
1349:  !---------------------------- ;
1350:  !Built PR[51] as OTF P[2] ;
1351:  R[270]=51    ;
1352:   ;
1353:  R[271]=57.943    ;
1354:  R[272]=382.104    ;
1355:  R[273]=300    ;
1356:  R[274]=(-170.927)    ;
1357:  R[275]=(-88.214)    ;
1358:  R[276]=(-7.494)    ;
1359:   ;
1360:  CALL CREATE_PR(R[270],R[271],R[272],R[273],R[274],R[275],R[276]) ;
1361:   ;
1362:  !---------------------------- ;
1363:  !Built PR[52] as OTF P[3] ;
1364:  R[280]=52    ;
1365:   ;
1366:  R[281]=58.385    ;
1367:  R[282]=833.481    ;
1368:  R[283]=300    ;
1369:  R[284]=(-171.562)    ;
1370:  R[285]=(-88.211)    ;
1371:  R[286]=(-7.433)    ;
1372:   ;
1373:  CALL CREATE_PR(R[280],R[281],R[282],R[283],R[284],R[285],R[286]) ;
1374:   ;
1375:  !Jump to end of the program ;
1376:  JMP LBL[9999] ;
1377:  !Template Ends ;
1378:   ;
1379:   ;
1380:  LBL[300] ;
1381:  !---------------------------- ;
1382:  !R[103]=300 -> "JOB_VAR_OD_GRIP" ;
1383:  !4By9 OTF Only, Max 144 piece ;
1384:  !Straight Face-plate Up/Down Pick ;
1385:  !---------------------------- ;
1386:  !Built PR[40] as Infeed P[1] ;
1387:  R[200]=40    ;
1388:   ;
1389:  R[201]=52.986    ;
1390:  R[202]=837.611    ;
1391:  R[203]=300    ;
1392:  R[204]=(-135.64)    ;
1393:  R[205]=(-89.334)    ;
1394:  R[206]=(-44.75)    ;
1395:   ;
1396:  CALL CREATE_PR(R[200],R[201],R[202],R[203],R[204],R[205],R[206]) ;
1397:   ;
1398:  !---------------------------- ;
1399:  !R[103]=300 -> "JOB_VAR_OD_GRIP" ;
1400:  !4By9 OTF Only, Max 144 piece ;
1401:  !Straight Face-plate Up/Down Pick ;
1402:  !---------------------------- ;
1403:  !Built PR[41] as Infeed P[2] ;
1404:  R[210]=41    ;
1405:   ;
1406:  R[211]=53.152    ;
1407:  R[212]=385.263    ;
1408:  R[213]=300    ;
1409:  R[214]=(-136.806)    ;
1410:  R[215]=(-89.315)    ;
1411:  R[216]=(-43.565)    ;
1412:   ;
1413:  CALL CREATE_PR(R[210],R[211],R[212],R[213],R[214],R[215],R[216]) ;
1414:   ;
1415:  !---------------------------- ;
1416:  !R[103]=300 -> "JOB_VAR_OD_GRIP" ;
1417:  !4By9 OTF Only, Max 144 piece ;
1418:  !Straight Face-plate Up/Down Pick ;
1419:  !---------------------------- ;
1420:  !Built PR[42] as Infeed P[3] ;
1421:  R[220]=42    ;
1422:   ;
1423:  R[221]=44.932    ;
1424:  R[222]=357.144    ;
1425:  R[223]=300    ;
1426:  R[224]=(-127.616)    ;
1427:  R[225]=(-89.079)    ;
1428:  R[226]=(-52.124)    ;
1429:   ;
1430:  CALL CREATE_PR(R[220],R[221],R[222],R[223],R[224],R[225],R[226]) ;
1431:   ;
1432:  !---------------------------- ;
1433:  !R[103]=300 -> "JOB_VAR_OD_GRIP" ;
1434:  !4By9 OTF Only, Max 144 piece ;
1435:  !Straight Face-plate Up/Down Pick ;
1436:  !---------------------------- ;
1437:  !Built PR[47] as Infeed P[4] ;
1438:  R[230]=47    ;
1439:   ;
1440:  R[231]=53.084    ;
1441:  R[232]=836.564    ;
1442:  R[233]=300    ;
1443:  R[234]=(-127.701)    ;
1444:  R[235]=(-89.072)    ;
1445:  R[236]=(-53.116)    ;
1446:   ;
1447:  CALL CREATE_PR(R[230],R[231],R[232],R[233],R[234],R[235],R[236]) ;
1448:   ;
1449:  !---------------------------- ;
1450:  !R[103]=300 -> "JOB_VAR_OD_GRIP" ;
1451:  !4By9 OTF Only, Max 144 piece ;
1452:  !Straight Face-plate Up/Down Pick ;
1453:  !---------------------------- ;
1454:  !Built PR[48] as Infeed P[5] ;
1455:  R[240]=48    ;
1456:   ;
1457:  R[241]=53.598    ;
1458:  R[242]=386.354    ;
1459:  R[243]=300    ;
1460:  R[244]=(-119.135)    ;
1461:  R[245]=(-89.246)    ;
1462:  R[246]=(-62.104)    ;
1463:   ;
1464:  CALL CREATE_PR(R[240],R[241],R[242],R[243],R[244],R[245],R[246]) ;
1465:   ;
1466:  !---------------------------- ;
1467:  !R[103]=300 -> "JOB_VAR_OD_GRIP" ;
1468:  !4By9 OTF Only, Max 144 piece ;
1469:  !Straight Face-plate Up/Down Pick ;
1470:  !---------------------------- ;
1471:  !Built PR[49] as Infeed P[6] ;
1472:  R[250]=49    ;
1473:   ;
1474:  R[251]=52.953    ;
1475:  R[252]=(-59.846)    ;
1476:  R[253]=300    ;
1477:  R[254]=(-123.722)    ;
1478:  R[255]=(-89.153)    ;
1479:  R[256]=(-57.497)    ;
1480:   ;
1481:  CALL CREATE_PR(R[250],R[251],R[252],R[253],R[254],R[255],R[256]) ;
1482:   ;
1483:  !---------------------------- ;
1484:  !R[103]=300 -> "JOB_VAR_OD_GRIP" ;
1485:  !4By9 OTF Only, Max 144 piece ;
1486:  !Straight Face-plate Up/Down Pick ;
1487:  !---------------------------- ;
1488:  !Built PR[50] as OTF P[1] ;
1489:  R[260]=50    ;
1490:   ;
1491:  R[261]=33.345    ;
1492:  R[262]=7.673    ;
1493:  R[263]=300    ;
1494:  R[264]=(-157.575)    ;
1495:  R[265]=(-88.384)    ;
1496:  R[266]=(-19.264)    ;
1497:   ;
1498:  CALL CREATE_PR(R[260],R[261],R[262],R[263],R[264],R[265],R[266]) ;
1499:   ;
1500:  !---------------------------- ;
1501:  !R[103]=300 -> "JOB_VAR_OD_GRIP" ;
1502:  !4By9 OTF Only, Max 144 piece ;
1503:  !Straight Face-plate Up/Down Pick ;
1504:  !---------------------------- ;
1505:  !Built PR[51] as OTF P[2] ;
1506:  R[270]=51    ;
1507:   ;
1508:  R[271]=40.956    ;
1509:  R[272]=296.424    ;
1510:  R[273]=300    ;
1511:  R[274]=(-157.514)    ;
1512:  R[275]=(-88.371)    ;
1513:  R[276]=(-19.346)    ;
1514:   ;
1515:  CALL CREATE_PR(R[270],R[271],R[272],R[273],R[274],R[275],R[276]) ;
1516:   ;
1517:  !---------------------------- ;
1518:  !R[103]=300 -> "JOB_VAR_OD_GRIP" ;
1519:  !4By9 OTF Only, Max 144 piece ;
1520:  !Straight Face-plate Up/Down Pick ;
1521:  !---------------------------- ;
1522:  !Built PR[52] as OTF P[3] ;
1523:  R[280]=52    ;
1524:   ;
1525:  R[281]=32.793    ;
1526:  R[282]=576.502    ;
1527:  R[283]=300    ;
1528:  R[284]=(-157.782)    ;
1529:  R[285]=(-88.365)    ;
1530:  R[286]=(-19.084)    ;
1531:   ;
1532:  CALL CREATE_PR(R[280],R[281],R[282],R[283],R[284],R[285],R[286]) ;
1533:   ;
1534:  !---------------------------- ;
1535:  !R[103]=300 -> "JOB_VAR_OD_GRIP" ;
1536:  !4By9 OTF Only, Max 144 piece ;
1537:  !Straight Face-plate Up/Down Pick ;
1538:  !---------------------------- ;
1539:  !Built PR[60] as OTF P[4] ;
1540:  R[290]=60    ;
1541:   ;
1542:  R[291]=33.089    ;
1543:  R[292]=862.155    ;
1544:  R[293]=300    ;
1545:  R[294]=(-157.966)    ;
1546:  R[295]=(-88.36)    ;
1547:  R[296]=(-18.903)    ;
1548:   ;
1549:  CALL CREATE_PR(R[290],R[291],R[292],R[293],R[294],R[295],R[296]) ;
1550:   ;
1551:  !Jump to end of the program ;
1552:  JMP LBL[9999] ;
1553:  !Template Ends ;
1554:   ;
1555:  LBL[320] ;
1556:   ;
1557:  !---------------------------- ;
1558:  !R[103]=320 -> "JOB_VAR_OD_GRIP" ;
1559:  !6By8 OTF Only, Max 144 piece ;
1560:  !Straight Face-plate Up/Down Pick ;
1561:  !---------------------------- ;
1562:  !Built PR[50] as OTF P[1] ;
1563:  R[260]=50    ;
1564:   ;
1565:  R[261]=33.345    ;
1566:  R[262]=7.673    ;
1567:  R[263]=300    ;
1568:  R[264]=(-157.575)    ;
1569:  R[265]=(-88.384)    ;
1570:  R[266]=(-19.264)    ;
1571:   ;
1572:  CALL CREATE_PR(R[260],R[261],R[262],R[263],R[264],R[265],R[266]) ;
1573:   ;
1574:  !---------------------------- ;
1575:  !R[103]=320 -> "JOB_VAR_OD_GRIP" ;
1576:  !6By8 OTF Only, Max 144 piece ;
1577:  !Straight Face-plate Up/Down Pick ;
1578:  !---------------------------- ;
1579:  !Built PR[51] as OTF P[2] ;
1580:  R[270]=51    ;
1581:   ;
1582:  R[271]=40.956    ;
1583:  R[272]=296.424    ;
1584:  R[273]=300    ;
1585:  R[274]=(-157.514)    ;
1586:  R[275]=(-88.371)    ;
1587:  R[276]=(-19.346)    ;
1588:   ;
1589:  CALL CREATE_PR(R[270],R[271],R[272],R[273],R[274],R[275],R[276]) ;
1590:   ;
1591:  !---------------------------- ;
1592:  !R[103]=320 -> "JOB_VAR_OD_GRIP" ;
1593:  !6By8 OTF Only, Max 144 piece ;
1594:  !Straight Face-plate Up/Down Pick ;
1595:  !---------------------------- ;
1596:  !Built PR[52] as OTF P[3] ;
1597:  R[280]=52    ;
1598:   ;
1599:  R[281]=32.793    ;
1600:  R[282]=576.502    ;
1601:  R[283]=300    ;
1602:  R[284]=(-157.782)    ;
1603:  R[285]=(-88.365)    ;
1604:  R[286]=(-19.084)    ;
1605:   ;
1606:  CALL CREATE_PR(R[280],R[281],R[282],R[283],R[284],R[285],R[286]) ;
1607:   ;
1608:  !Jump to end of the program ;
1609:  JMP LBL[9999] ;
1610:  !Template Ends ;
1611:   ;
1612:  LBL[340] ;
1613:  !---------------------------- ;
1614:  !R[103]=340 -> "JOB_VAR_OD_GRIP" ;
1615:  !3By4 INF OD-GRIP, Max 36 piece ;
1616:  !BOX Up/Down Pick ;
1617:  !---------------------------- ;
1618:  !Built PR[40] as Infeed P[1] ;
1619:  R[200]=40    ;
1620:   ;
1621:  R[201]=77.044    ;
1622:  R[202]=825.268    ;
1623:  R[203]=149.376    ;
1624:  R[204]=20.058    ;
1625:  R[205]=(-88.647)    ;
1626:  R[206]=160.787    ;
1627:   ;
1628:  CALL CREATE_PR(R[200],R[201],R[202],R[203],R[204],R[205],R[206]) ;
1629:   ;
1630:  !---------------------------- ;
1631:  !R[103]=340 -> "JOB_VAR_OD_GRIP" ;
1632:  !3By4 INF OD-GRIP, Max 36 piece ;
1633:  !BOX Up/Down Pick ;
1634:  !---------------------------- ;
1635:  !Built PR[41] as Infeed P[2] ;
1636:  R[210]=41    ;
1637:   ;
1638:  R[211]=73.737    ;
1639:  R[212]=373.59    ;
1640:  R[213]=146.101    ;
1641:  R[214]=20.623    ;
1642:  R[215]=(-88.685)    ;
1643:  R[216]=160.248    ;
1644:   ;
1645:  CALL CREATE_PR(R[210],R[211],R[212],R[213],R[214],R[215],R[216]) ;
1646:   ;
1647:  !---------------------------- ;
1648:  !R[103]=340 -> "JOB_VAR_OD_GRIP" ;
1649:  !3By4 INF OD-GRIP, Max 36 piece ;
1650:  !BOX Up/Down Pick ;
1651:  !---------------------------- ;
1652:  !Built PR[42] as Infeed P[3] ;
1653:  R[220]=42    ;
1654:   ;
1655:  R[221]=75.997    ;
1656:  R[222]=(-75.158)    ;
1657:  R[223]=162.092    ;
1658:  R[224]=20.675    ;
1659:  R[225]=(-88.731)    ;
1660:  R[226]=160.229    ;
1661:   ;
1662:  CALL CREATE_PR(R[220],R[221],R[222],R[223],R[224],R[225],R[226]) ;
1663:   ;
1664:  !---------------------------- ;
1665:  !R[103]=340 -> "JOB_VAR_OD_GRIP" ;
1666:  !3By4 INF OD-GRIP, Max 36 piece ;
1667:  !BOX Up/Down Pick ;
1668:  !---------------------------- ;
1669:  !Built PR[50] as OTF P[1] ;
1670:  R[230]=50    ;
1671:   ;
1672:  R[231]=66.596    ;
1673:  R[232]=(-72.932)    ;
1674:  R[233]=700    ;
1675:  R[234]=5.353    ;
1676:  R[235]=(-88.806)    ;
1677:  R[236]=173.83    ;
1678:   ;
1679:  CALL CREATE_PR(R[230],R[231],R[232],R[233],R[234],R[235],R[236]) ;
1680:   ;
1681:  !---------------------------- ;
1682:  !R[103]=340 -> "JOB_VAR_OD_GRIP" ;
1683:  !3By4 INF OD-GRIP, Max 36 piece ;
1684:  !BOX Up/Down Pick ;
1685:  !---------------------------- ;
1686:  !Built PR[51] as OTF P[2] ;
1687:  R[240]=51    ;
1688:   ;
1689:  R[241]=70.095    ;
1690:  R[242]=378.905    ;
1691:  R[243]=700    ;
1692:  R[244]=(-4.178)    ;
1693:  R[245]=(-88.742)    ;
1694:  R[246]=(-176.605)    ;
1695:   ;
1696:  CALL CREATE_PR(R[240],R[241],R[242],R[243],R[244],R[245],R[246]) ;
1697:   ;
1698:  !---------------------------- ;
1699:  !R[103]=340 -> "JOB_VAR_OD_GRIP" ;
1700:  !3By4 INF OD-GRIP, Max 36 piece ;
1701:  !BOX Up/Down Pick ;
1702:  !---------------------------- ;
1703:  !Built PR[52] as OTF P[3] ;
1704:  R[250]=52    ;
1705:   ;
1706:  R[251]=70.211    ;
1707:  R[252]=829.862    ;
1708:  R[253]=700    ;
1709:  R[254]=(-7.014)    ;
1710:  R[255]=(-88.859)    ;
1711:  R[256]=(-173.67)    ;
1712:   ;
1713:  CALL CREATE_PR(R[250],R[251],R[252],R[253],R[254],R[255],R[256]) ;
1714:   ;
1715:  !Jump to end of the program ;
1716:  JMP LBL[9999] ;
1717:  !Template Ends ;
1718:  !---------------------------- ;
1719:  LBL[9999:END] ;
1720:  END ;
/POS
/END
